// TIA Portal V19 export
TYPE "lexchangetray_typeroller_signalTM_Simulation"
// Type: Bool
// stored: Access Published
   STRUCT
      trayAutomaticDischargeDetectionEm1 : Bool;   // Manual mode parameters for axis control interface
      trayAutomaticFeedingDetectionEm1 : Bool;   // Manual mode parameters for axis control interface
      restraintTrayAntiReverseDetection2Em1 : Bool;   // Manual mode parameters for axis control interface
      restraintTrayAntiReverseDetection1Em1 : Bool;   // Manual mode parameters for axis control interface
   END_STRUCT;
END_TYPE
